{attribute 'qualified_only'}
VAR_GLOBAL
	
//Atrium
	strEnOceanSwitch_AtriumNiveau_PladeB				: Tc2_EnOcean.STR_EnOceanSwitch;
	strEnOceanSwitch_AtriumNiveau_Service				: Tc2_EnOcean.STR_EnOceanSwitch;


//Gange
//	strEnOceanSwitch_Gang_3_364				: Tc2_EnOcean.STR_EnOceanSwitch;

	//
 
     strEnOceanSwitch_Rum_3_529                      	: Tc2_EnOcean.STR_EnOceanSwitch;


END_VAR

(* stored: Version 1.1.0.1
   GVL GVL_EnOcean: Id {bec68ff9-8f1d-4ce1-b8b9-84de691aacc9} *)
